FUNCTION_BLOCK FB_SafeDiag
VAR_INPUT
END_VAR
VAR_OUTPUT
END_VAR
VAR
END_VAR

END_FUNCTION_BLOCK

(* stored: Version 1.1.0.1, ProductVersion 3.1.4024.11
   POU FB_SafeDiag: Id {28431db4-d0e1-073b-2ee2-e5cdfa2aa643}, SpecialFunc None *)
